PROGRAM MAIN
VAR
	RealSingleton	: FB_Singleton;
	Singleton		: POINTER TO FB_Singleton;
	populate		: BOOL;
END_VAR

Singleton := RealSingleton.Instance;

IF populate THEN
	Singleton^.AddAlarm('Populated from main pou');
	populate := FALSE;
END_IF

SecondPou();

END_PROGRAM

(* stored: Version 1.1.0.1, ProductVersion 3.1.4024.12
   POU MAIN: Id {d0ba762e-8cde-4cd2-a9ff-650b6e34056b}, SpecialFunc None *)
